TYPE ST_BigBagActualMassStoreOutValues :
STRUCT
    rBagActualMass : REAL; // aktualna masa worka jako jedno źródło prawdy
END_STRUCT
END_TYPE

(* stored: Version 1.1.0.1, ProductVersion 3.1.4024.16
   DUT ST_BigBagActualMassStoreOutValues: Id {f763a921-cae9-4706-9f3b-f26d446521e9} *)
